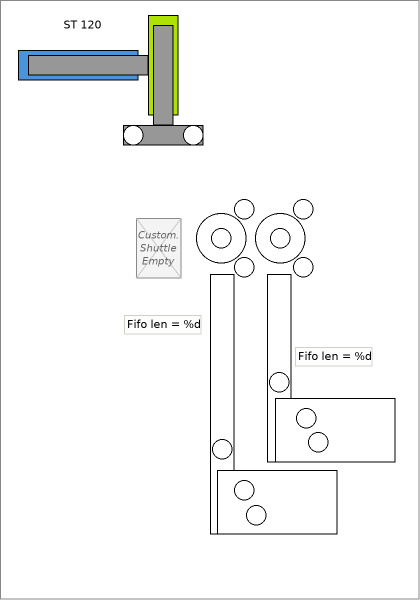
VISUALIZATION VISU_ST120  // 420x600
    Ellipse (196,213 50x50), colour toggle: GVL._Process4.fb_Feeder.fb_pivotLeft.xOUT_VALVE
    Image (136,218 45x60), invisible if: NOT __ISVALIDREF(GVL._Process4._Mover), image: Custom.Shuttle Empty
    Rectangle (18,50 120x30)
    Rectangle (28,55 120x20)
        p3560616238: GVL._Process4.fb_Pnp.fb_simu_axis120_01Y.rOUT_PixActual
    Rectangle (148,15 30x100)
        p3560616238: GVL._Process4.fb_Pnp.fb_simu_axis120_01Y.rOUT_PixActual
    Rectangle (153,25 20x100)
        p2738717112: GVL._Process4.fb_Pnp.fb_simu_axis120_02Z.rOUT_PixActual
        p3560616238: GVL._Process4.fb_Pnp.fb_simu_axis120_01Y.rOUT_PixActual
    Rectangle (210,274 24x260)
    Ellipse (212,439 20x20), colour toggle: GVL._Process4.fb_Feeder.simu_fifoLeft.IsFull()
    Ellipse (211,228 20x20), colour toggle: GVL._Process4.fb_Feeder.simu_fifoLeft.IsFull()
    Textfield (124,315 77x19), "Fifo len = %d", text variable: GVL._Process4.fb_Feeder.simu_fifoLeft.GetLen()
    Label (40,15 85x20), "ST 120"
    RoundedRectangle (217,470 120x64), colour toggle: GVL._Process4.fb_Feeder.fb_feederLeft.xOUT_EnableFeeder
    Rectangle (267,274 24x188)
    Ellipse (269,372 20x20), colour toggle: GVL._Process4.fb_Feeder.simu_fifoRight.IsFull()
    RoundedRectangle (275,398 120x64), colour toggle: GVL._Process4.fb_Feeder.fb_feederRight.xOUT_EnableFeeder
    Rectangle (123,125 80x20)
        p2738717112: GVL._Process4.fb_Pnp.fb_simu_axis120_02Z.rOUT_PixActual
        p3560616238: GVL._Process4.fb_Pnp.fb_simu_axis120_01Y.rOUT_PixActual
    Ellipse (183,125 20x20), colour toggle: GVL._Process4.fb_Pnp.fb_gripperRight.xIN_AS
        p3560616238: GVL._Process4.fb_Pnp.fb_simu_axis120_01Y.rOUT_PixActual
        p2738717112: GVL._Process4.fb_Pnp.fb_simu_axis120_02Z.rOUT_PixActual
    Ellipse (123,125 20x20), colour toggle: GVL._Process4.fb_Pnp.fb_gripperLeft.xIN_AS
        p3560616238: GVL._Process4.fb_Pnp.fb_simu_axis120_01Y.rOUT_PixActual
        p2738717112: GVL._Process4.fb_Pnp.fb_simu_axis120_02Z.rOUT_PixActual
    Textfield (295,347 77x19), "Fifo len = %d", text variable: GVL._Process4.fb_Feeder.simu_fifoRight.GetLen()
    Ellipse (255,213 50x50), colour toggle: GVL._Process4.fb_Feeder.fb_pivotRight.xOUT_VALVE
    Ellipse (270,228 20x20), colour toggle: GVL._Process4.fb_Feeder.simu_fifoRight.IsFull()
    Ellipse (293,199 20x20), colour toggle: GVL._Process4.fb_Feeder.fb_pivotRight.xIN_GS
    Ellipse (293,257 20x20), colour toggle: GVL._Process4.fb_Feeder.fb_pivotRight.xIN_AS
    Ellipse (234,199 20x20), colour toggle: GVL._Process4.fb_Feeder.fb_pivotLeft.xIN_GS
    Ellipse (234,257 20x20), colour toggle: GVL._Process4.fb_Feeder.fb_pivotLeft.xIN_AS
    Ellipse (246,505 20x20), colour toggle: GVL._Process4.fb_Feeder.fb_hubladerLeft.xIN_GS
    Ellipse (234,480 20x20), colour toggle: GVL._Process4.fb_Feeder.fb_hubladerLeft.xIN_AS
    Ellipse (296,408 20x20), colour toggle: GVL._Process4.fb_Feeder.fb_hubladerRight.xIN_AS
    Ellipse (308,432 20x20), colour toggle: GVL._Process4.fb_Feeder.fb_hubladerRight.xIN_GS
END_VISUALIZATION

(* stored: Version 1.1.0.1, ProductVersion 3.1.4024.6
   Visu VISU_ST120: Id {7a29c01d-e6f4-44b4-bc7e-5918cebc9b69} *)
